(* PLC project 1st_testSTEPPER_SFL3, BrAutomation SafeDESIGNER  5.12.2.0 *)
(* stored: companyURL http://www.br-automation.com, creationDateTime Wed Mar 31 14:59:11 2021 *)

PROGRAM Main

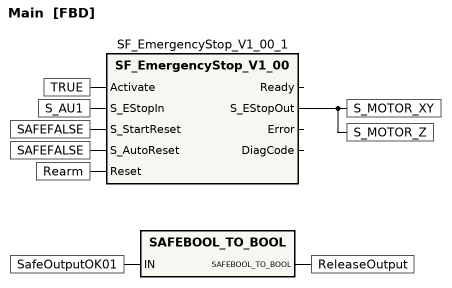
(* FBD diagram, written out as Structured Text *)
ReleaseOutput := SAFEBOOL_TO_BOOL(SafeOutputOK01);
SF_EmergencyStop_V1_00_1(Activate := TRUE, S_EStopIn := S_AU1, S_StartReset := SAFEFALSE, S_AutoReset := SAFEFALSE, Reset := Rearm);
S_MOTOR_XY := SF_EmergencyStop_V1_00_1.S_EStopOut;
S_MOTOR_Z := SF_EmergencyStop_V1_00_1.S_EStopOut;
END_PROGRAM
